// TIA Portal project "Function Block Pusher" (V16)
// Vorlageprojekt für das Buch mit Zielsystem S7-1200

(* hardware
DEVICE "S7-1200-Station_1"  S7-1200 Station
   slot 0: "Baugruppenträger_0"  Rack  V1.0
   slot 1: "PLC_1"  CPU 1211C DC/DC/DC  6ES7 211-1AE40-0XB0  V4.1
*)

// ===== PLC "PLC_1"  CPU 1211C DC/DC/DC =====

VAR_GLOBAL   // PLC tag table "Standard-Variablentabelle"
   "xStatstart" AT %M0.6 : Bool;
   "xMem" AT %M0.7 : Bool;
   "xAlarmstat" AT %M1.0 : Bool;
   "xstep_0" AT %M1.1 : Bool;
   "xstep_10" AT %M1.2 : Bool;
   "xstep_20" AT %M1.3 : Bool;
   "xstep_30" AT %M1.4 : Bool;
   "xAlarm" AT %M1.5 : Bool;
   "xReset" AT %M1.6 : Bool;
END_VAR

VAR_GLOBAL   // PLC tag table "Tag table_1"
   "xPusherSensFront_1" AT %I0.1 : Bool;
   "xPusherSensBck_1" AT %I0.0 : Bool;
   "xPusherSensFront_2" AT %I0.3 : Bool;
   "xPusherSensBck_2" AT %I0.2 : Bool;
   "xPusherSensFront_3" AT %I0.5 : Bool;
   "xPusherSensBck_3" AT %I0.4 : Bool;
   "xStart" AT %I0.6 : Bool;
   "xStop" AT %I0.7 : Bool;
   "xPusherCoil_1" AT %Q0.0 : Bool;
   "xPusherCoil_2" AT %Q0.1 : Bool;
   "xPusherCoil_3" AT %Q0.2 : Bool;
   "xStartLed" AT %Q0.3 : Bool;
   "xStopLed" AT %Q0.4 : Bool;
   "xAlarmLed" AT %Q0.5 : Bool;
END_VAR

DATA_BLOCK "instPusherMain"   // DB1
{ S7_Optimized_Access := 'TRUE' }
VERSION : 0.1
// stored: InstanceOfName FB_Pusher
"FB_Pusher"
BEGIN
END_DATA_BLOCK

DATA_BLOCK "instPusherMain0"   // DB2
{ S7_Optimized_Access := 'TRUE' }
VERSION : 0.1
// stored: InstanceOfName FB_Pusher
"FB_Pusher"
BEGIN
END_DATA_BLOCK

DATA_BLOCK "instPusherMain2"   // DB3
{ S7_Optimized_Access := 'TRUE' }
VERSION : 0.1
// stored: InstanceOfName FB_Pusher
"FB_Pusher"
BEGIN
END_DATA_BLOCK

DATA_BLOCK "instPusherMain1"   // DB4
{ S7_Optimized_Access := 'TRUE' }
VERSION : 0.1
// stored: InstanceOfName FB_Pusher
"FB_Pusher"
BEGIN
END_DATA_BLOCK

// folder: System blocks/Program resources

DATA_BLOCK "IEC_Timer_0_DB"   // DB5
{ S7_Optimized_Access := 'TRUE' }
AUTHOR : Simatic
FAMILY : IEC
NAME : IEC_TMR
VERSION : 1.0
// stored: InstanceOfName IEC_TIMER
"IEC_TIMER"
BEGIN
END_DATA_BLOCK

// folder: (top level)

FUNCTION_BLOCK "FB_Pusher"   // FB1, LAD
{ S7_Optimized_Access := 'TRUE' }
VERSION : 0.1
   VAR_INPUT
      xExtend : Bool;
      xSensorBck : Bool;
      xSensorFront : Bool;
   END_VAR
   VAR_OUTPUT
      xPosBck : Bool;
      xPosFront : Bool;
      XAlarm : Bool;
      xCoil : Bool;
   END_VAR
   VAR
      IEC_Timer_0_Instance : TON_TIME;
   END_VAR
   VAR RETAIN
      "dicycle Cnt" : DInt;
   END_VAR
   VAR CONSTANT
      timeAlarm_TIME : Time := T#3s;
   END_VAR
BEGIN

REGION Network 1
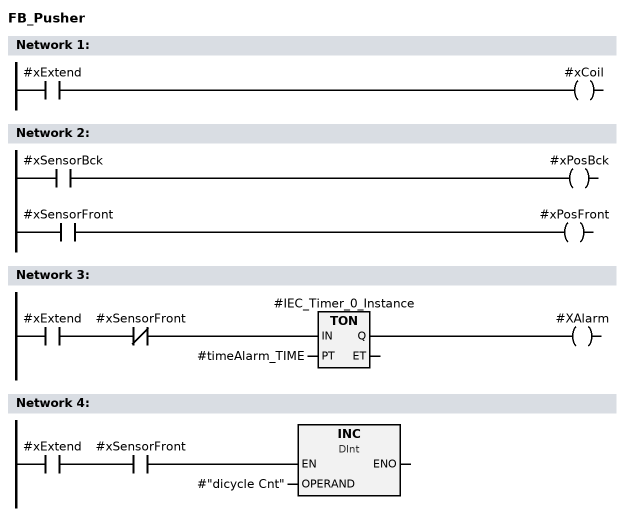
   RUNG wire#powerrail
      Contact( #xExtend )
      Coil( #xCoil )
   END_RUNG
   // the same network as SCL:
   #xCoil := #xExtend;
END_REGION

REGION Network 2
   RUNG wire#powerrail
      Contact( #xSensorBck )
      Coil( #xPosBck )
   END_RUNG
   RUNG wire#powerrail
      Contact( #xSensorFront )
      Coil( #xPosFront )
   END_RUNG
   // the same network as SCL:
   #xPosBck := #xSensorBck;
   #xPosFront := #xSensorFront;
END_REGION

REGION Network 3
   #IEC_Timer_0_Instance(IN := #xExtend AND NOT #xSensorFront, PT := #timeAlarm_TIME);   // TON
   #XAlarm := #IEC_Timer_0_Instance.Q;
END_REGION

REGION Network 4
   RUNG wire#powerrail
      Contact( #xExtend )
      Contact( #xSensorFront )
      { S7_Templates := "DestType := DInt" } Inc( #"dicycle Cnt" )
   END_RUNG
   // the same network as SCL:
   IF #xExtend AND #xSensorFront THEN #"dicycle Cnt" := #"dicycle Cnt" + 1; END_IF;
END_REGION
END_FUNCTION_BLOCK

FUNCTION "MHJ-PLC-Lab-Function-S71200" : Void   // FC9000, SCL
{ S7_Optimized_Access := 'TRUE' }
VERSION : 0.1
   VAR_TEMP
      rdTimeReturn : Int;
      outputTime : DTL;
      SyncVal : Byte;
      forVal : Int;
      forVal_2 : Int;
      Value : Byte;
   END_VAR
   VAR CONSTANT
      CompVal : Byte := 16#34;
      Value_01 : Byte := 16#11;
      Value_01_DW : DWord := 16#A165_D992;
      Value_02_DW : DWord := 16#58BE_4401;
   END_VAR
BEGIN

   #Value:=PEEK(area := 16#82,
        dbNumber := 0,
        byteOffset := 511);
   #Value := #Value + 1;

   POKE(area := 16#82,
        dbNumber := 0,
        byteOffset := 511,
        value := #Value);

   POKE(area:=16#81,
        dbNumber:=0,
        byteOffset:=1016,
        value:=#Value_01_DW);
   POKE(area := 16#81,
        dbNumber := 0,
        byteOffset := 1020,
        value := #Value_02_DW);

   POKE(area := 16#81,
        dbNumber := 0,
        byteOffset := 511,
        value := B#16#00);

   FOR #forVal := 0 TO 120 DO
       FOR #forVal_2:=0 TO 10 DO
           #rdTimeReturn:=RD_SYS_T(#outputTime);
           #rdTimeReturn := WR_SYS_T(#outputTime);
           #rdTimeReturn := RD_SYS_T(#outputTime);
           #rdTimeReturn := WR_SYS_T(#outputTime);
       END_FOR;
       #SyncVal:= PEEK(area := 16#81,
                      dbNumber := 0,
                      byteOffset := 511);
       IF #SyncVal = #CompVal THEN
          GOTO M_1;
       END_IF;
   END_FOR;
   RETURN;

   M_1:
   POKE(area := 16#81,
        dbNumber := 0,
        byteOffset := 511,
        value := B#16#0);
END_FUNCTION

ORGANIZATION_BLOCK "Main"   // OB1, LAD, ProgramCycle
TITLE = "Main Program Sweep (Cycle)"
{ S7_Optimized_Access := 'TRUE' }
VERSION : 0.1
   VAR_INPUT
      Initial_Call : Bool;   // Initial call of this OB
      Remanence : Bool;   // =True, if remanent data are available
   END_VAR
   VAR_TEMP   // added for the SCL form of the ladder/FBD networks
      _w1 : Bool;
      _w2 : Bool;
   END_VAR
BEGIN

REGION Network 1
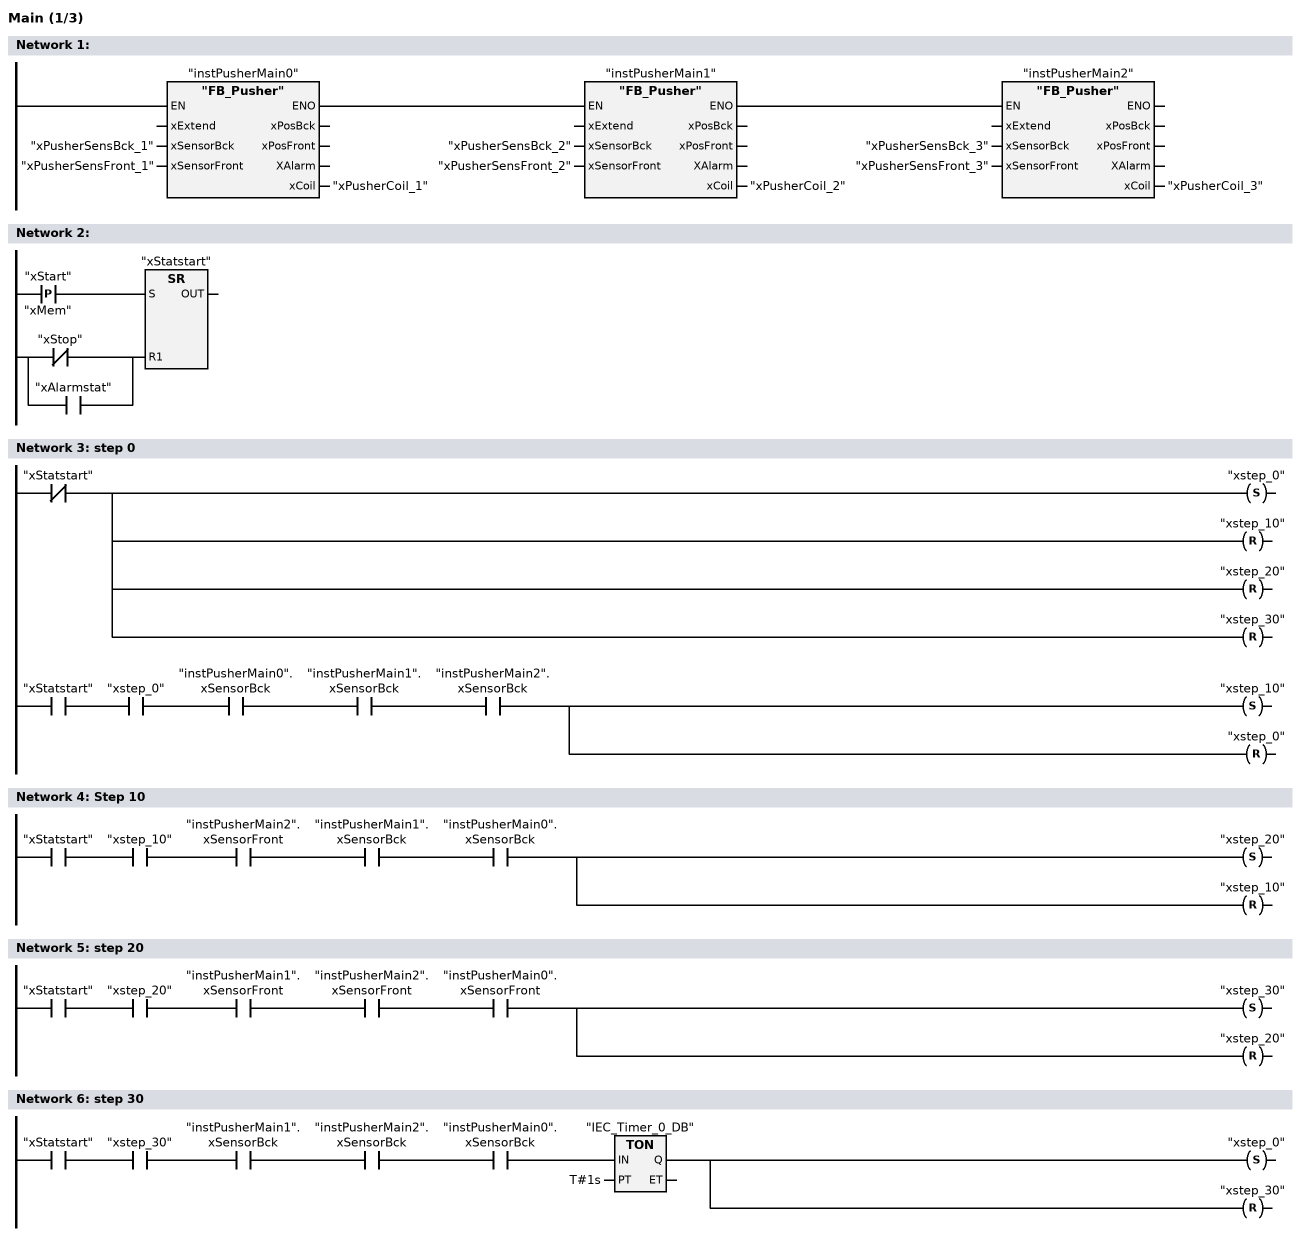
   RUNG wire#powerrail
      "instPusherMain0"(xExtend :=, xSensorBck := "xPusherSensBck_1", xSensorFront := "xPusherSensFront_1", xPosBck =>, xPosFront =>, XAlarm =>, xCoil => "xPusherCoil_1")
      "instPusherMain1"(xExtend :=, xSensorBck := "xPusherSensBck_2", xSensorFront := "xPusherSensFront_2", xPosBck =>, xPosFront =>, XAlarm =>, xCoil => "xPusherCoil_2")
      "instPusherMain2"(xExtend :=, xSensorBck := "xPusherSensBck_3", xSensorFront := "xPusherSensFront_3", xPosBck =>, xPosFront =>, XAlarm =>, xCoil => "xPusherCoil_3")
   END_RUNG
   // the same network as SCL:
   "instPusherMain0"(xSensorBck := "xPusherSensBck_1",   // "FB_Pusher"
                     xSensorFront := "xPusherSensFront_1",
                     xCoil => "xPusherCoil_1",
                     ENO => #_w1);
   "instPusherMain1"(EN := #_w1,   // "FB_Pusher"
                     xSensorBck := "xPusherSensBck_2",
                     xSensorFront := "xPusherSensFront_2",
                     xCoil => "xPusherCoil_2",
                     ENO => #_w2);
   IF #_w2 THEN
       "instPusherMain2"(xSensorBck := "xPusherSensBck_3",   // "FB_Pusher"
                         xSensorFront := "xPusherSensFront_3",
                         xCoil => "xPusherCoil_3");
   END_IF;
END_REGION

REGION Network 2
   RUNG wire#powerrail
      P_Contact(operand := "xStart", bit := "xMem")
      S_SR(operand := "xStatstart", r1 := wire#w1)
   END_RUNG
   RUNG wire#powerrail
      I_Contact( "xStop" )
   END_RUNG wire#w1
   RUNG wire#powerrail
      Contact( "xAlarmstat" )
   END_RUNG wire#w1
   // the same network as SCL:
   #_w1 := "xStart" AND NOT "xMem";   // rising edge of "xStart"
   "xMem" := "xStart";
   IF #_w1 THEN
       "xStatstart" := TRUE;   // SR flip-flop
   END_IF;
   IF NOT "xStop" OR "xAlarmstat" THEN "xStatstart" := FALSE; END_IF;
END_REGION

REGION Network 3: step 0
   RUNG wire#powerrail
      I_Contact( "xStatstart" )
      wire#w1
      S_Coil( "xstep_0" )
   END_RUNG
   RUNG wire#w1
      R_Coil( "xstep_10" )
   END_RUNG
   RUNG wire#w1
      R_Coil( "xstep_20" )
   END_RUNG
   RUNG wire#w1
      R_Coil( "xstep_30" )
   END_RUNG
   RUNG wire#powerrail
      Contact( "xStatstart" )
      Contact( "xstep_0" )
      Contact( "instPusherMain0".xSensorBck )
      Contact( "instPusherMain1".xSensorBck )
      Contact( "instPusherMain2".xSensorBck )
      wire#w2
      S_Coil( "xstep_10" )
   END_RUNG
   RUNG wire#w2
      R_Coil( "xstep_0" )
   END_RUNG
   // the same network as SCL:
   IF NOT "xStatstart" THEN
       "xstep_0" := TRUE;
       "xstep_10" := FALSE;
       "xstep_20" := FALSE;
       "xstep_30" := FALSE;
   END_IF;
   IF "xStatstart" AND "xstep_0" AND "instPusherMain0".xSensorBck AND "instPusherMain1".xSensorBck AND "instPusherMain2".xSensorBck THEN
       "xstep_10" := TRUE;
       "xstep_0" := FALSE;
   END_IF;
END_REGION

REGION Network 4: Step 10
   RUNG wire#powerrail
      Contact( "xStatstart" )
      Contact( "xstep_10" )
      Contact( "instPusherMain2".xSensorFront )
      Contact( "instPusherMain1".xSensorBck )
      Contact( "instPusherMain0".xSensorBck )
      wire#w1
      S_Coil( "xstep_20" )
   END_RUNG
   RUNG wire#w1
      R_Coil( "xstep_10" )
   END_RUNG
   // the same network as SCL:
   IF "xStatstart" AND "xstep_10" AND "instPusherMain2".xSensorFront AND "instPusherMain1".xSensorBck AND "instPusherMain0".xSensorBck THEN
       "xstep_20" := TRUE;
       "xstep_10" := FALSE;
   END_IF;
END_REGION

REGION Network 5: step 20
   RUNG wire#powerrail
      Contact( "xStatstart" )
      Contact( "xstep_20" )
      Contact( "instPusherMain1".xSensorFront )
      Contact( "instPusherMain2".xSensorFront )
      Contact( "instPusherMain0".xSensorFront )
      wire#w1
      S_Coil( "xstep_30" )
   END_RUNG
   RUNG wire#w1
      R_Coil( "xstep_20" )
   END_RUNG
   // the same network as SCL:
   IF "xStatstart" AND "xstep_20" AND "instPusherMain1".xSensorFront AND "instPusherMain2".xSensorFront AND "instPusherMain0".xSensorFront THEN
       "xstep_30" := TRUE;
       "xstep_20" := FALSE;
   END_IF;
END_REGION

REGION Network 6: step 30
   "IEC_Timer_0_DB".TON(IN := "xStatstart" AND "xstep_30" AND "instPusherMain1".xSensorBck AND "instPusherMain2".xSensorBck AND "instPusherMain0".xSensorBck,
                        PT := T#1s);
   IF "IEC_Timer_0_DB".Q THEN
       "xstep_0" := TRUE;
       "xstep_30" := FALSE;
   END_IF;
END_REGION

REGION Network 7
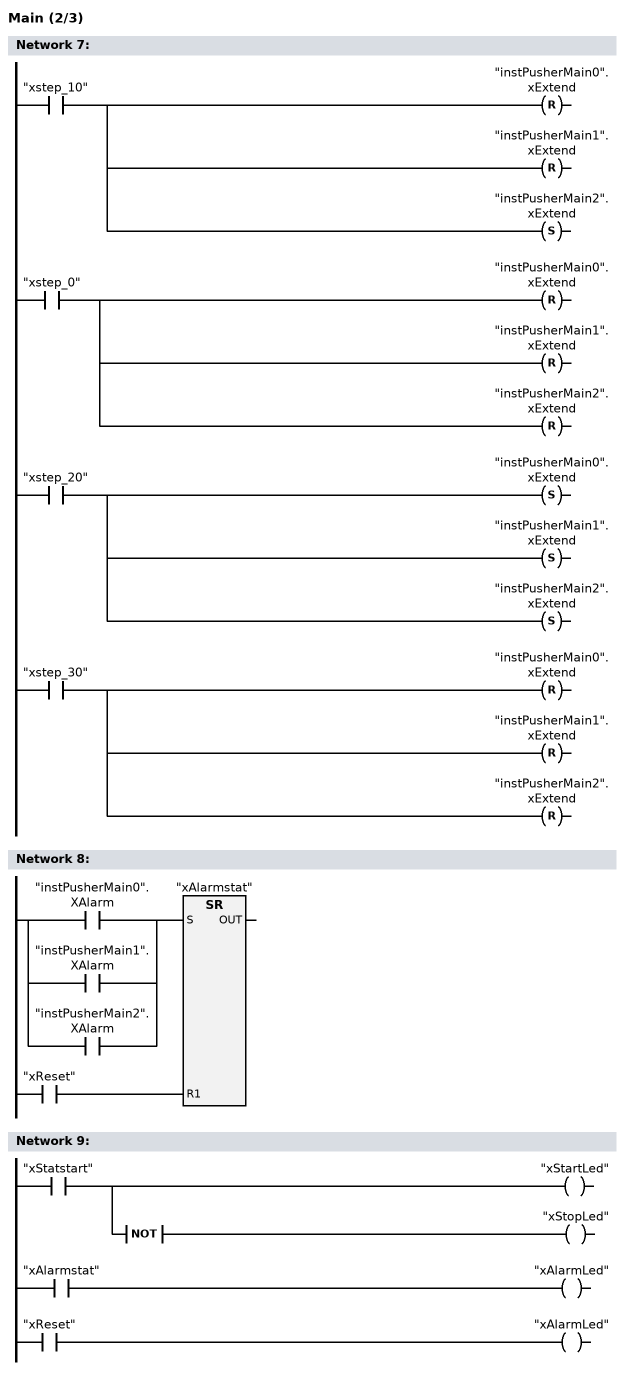
   RUNG wire#powerrail
      Contact( "xstep_10" )
      wire#w1
      R_Coil( "instPusherMain0".xExtend )
   END_RUNG
   RUNG wire#w1
      R_Coil( "instPusherMain1".xExtend )
   END_RUNG
   RUNG wire#w1
      S_Coil( "instPusherMain2".xExtend )
   END_RUNG
   RUNG wire#powerrail
      Contact( "xstep_0" )
      wire#w2
      R_Coil( "instPusherMain0".xExtend )
   END_RUNG
   RUNG wire#w2
      R_Coil( "instPusherMain1".xExtend )
   END_RUNG
   RUNG wire#w2
      R_Coil( "instPusherMain2".xExtend )
   END_RUNG
   RUNG wire#powerrail
      Contact( "xstep_20" )
      wire#w3
      S_Coil( "instPusherMain0".xExtend )
   END_RUNG
   RUNG wire#w3
      S_Coil( "instPusherMain1".xExtend )
   END_RUNG
   RUNG wire#w3
      S_Coil( "instPusherMain2".xExtend )
   END_RUNG
   RUNG wire#powerrail
      Contact( "xstep_30" )
      wire#w4
      R_Coil( "instPusherMain0".xExtend )
   END_RUNG
   RUNG wire#w4
      R_Coil( "instPusherMain1".xExtend )
   END_RUNG
   RUNG wire#w4
      R_Coil( "instPusherMain2".xExtend )
   END_RUNG
   // the same network as SCL:
   IF "xstep_10" THEN
       "instPusherMain0".xExtend := FALSE;
       "instPusherMain1".xExtend := FALSE;
       "instPusherMain2".xExtend := TRUE;
   END_IF;
   IF "xstep_0" THEN
       "instPusherMain0".xExtend := FALSE;
       "instPusherMain1".xExtend := FALSE;
       "instPusherMain2".xExtend := FALSE;
   END_IF;
   IF "xstep_20" THEN
       "instPusherMain0".xExtend := TRUE;
       "instPusherMain1".xExtend := TRUE;
       "instPusherMain2".xExtend := TRUE;
   END_IF;
   IF "xstep_30" THEN
       "instPusherMain0".xExtend := FALSE;
       "instPusherMain1".xExtend := FALSE;
       "instPusherMain2".xExtend := FALSE;
   END_IF;
END_REGION

REGION Network 8
   RUNG wire#powerrail
      Contact( "instPusherMain0".XAlarm )
      wire#w1
      S_SR(operand := "xAlarmstat", r1 := wire#w2)
   END_RUNG
   RUNG wire#powerrail
      Contact( "instPusherMain1".XAlarm )
   END_RUNG wire#w1
   RUNG wire#powerrail
      Contact( "instPusherMain2".XAlarm )
   END_RUNG wire#w1
   RUNG wire#powerrail
      Contact( "xReset" )
   END_RUNG wire#w2
   // the same network as SCL:
   IF "instPusherMain0".XAlarm OR "instPusherMain1".XAlarm OR "instPusherMain2".XAlarm THEN
       "xAlarmstat" := TRUE;   // SR flip-flop
   END_IF;
   IF "xReset" THEN "xAlarmstat" := FALSE; END_IF;
END_REGION

REGION Network 9
   RUNG wire#powerrail
      Contact( "xStatstart" )
      wire#w1
      Coil( "xStartLed" )
   END_RUNG
   RUNG wire#w1
      Not()
      Coil( "xStopLed" )
   END_RUNG
   RUNG wire#powerrail
      Contact( "xAlarmstat" )
      Coil( "xAlarmLed" )
   END_RUNG
   RUNG wire#powerrail
      Contact( "xReset" )
      Coil( "xAlarmLed" )
   END_RUNG
   // the same network as SCL:
   "xStartLed" := "xStatstart";
   "xStopLed" := NOT "xStatstart";
   "xAlarmLed" := "xAlarmstat";
   "xAlarmLed" := "xReset";
END_REGION

REGION Network 10
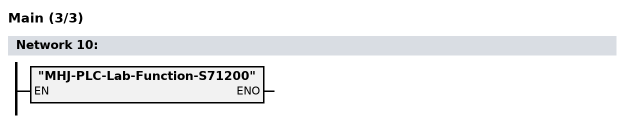
   RUNG wire#powerrail
      "MHJ-PLC-Lab-Function-S71200"()
   END_RUNG
   // the same network as SCL:
   "MHJ-PLC-Lab-Function-S71200"();
END_REGION
END_ORGANIZATION_BLOCK